RoboDK station: pega_analisa_e_posiciona.rdk

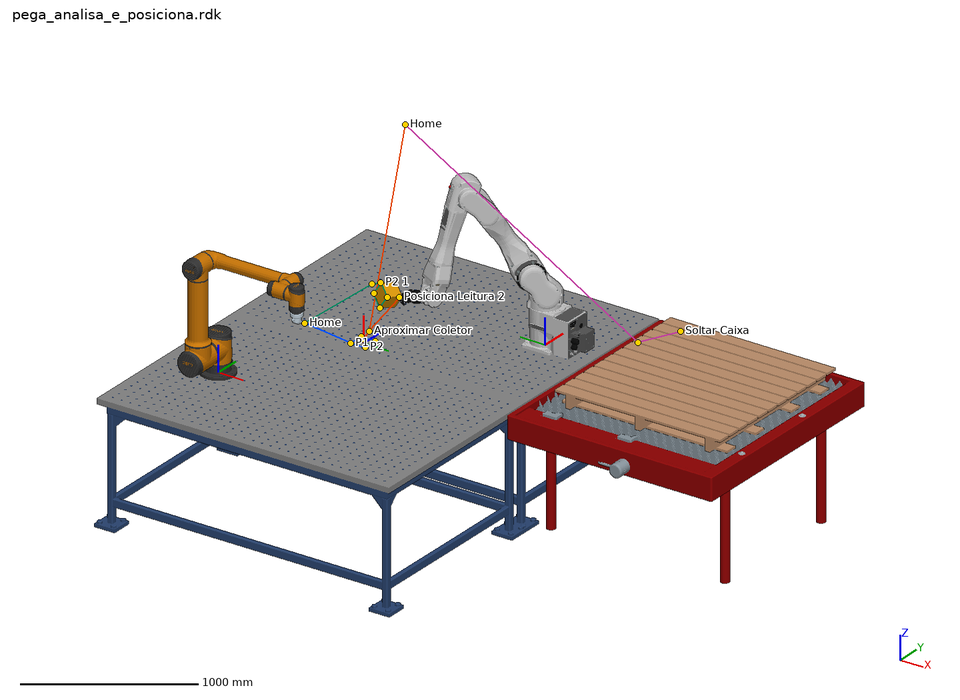
[picture v0: the station drawn from its stored meshes, robots at their saved joint values, targets as dots, program paths as lines]
Station pega_analisa_e_posiciona (saved by RoboDK 6.0.4). Poses are relative to the parent item; angles as X-Y-Z fixed-axis rotations.
  - frame Frame 3 at (0, 2000, 0) mm
    - object Table 2000x1200x800mm at (0, 1320, 0) mm, size 2020 x 1340 x 800 mm, geometry from Table-2000x1200x800mm.sld
    - frame Epson C12XL-A1401 Base at (1300, 1340, 0) mm, rotated rx 0 ry 0 rz 90 deg
      - robot Epson C12XL-A1401: 6 axes, payload 12 kg, reach 1400 mm, repeatability 0.05 mm, weight 63 kg
          modified DH rows (alpha deg, a mm, theta deg, d mm): 0, 0, 0, 472; -90, 100, -90, 0; 0, 650, 0, 0; -90, 30, 0, 650; 90, 0, 0, 0; -90, 0, 0, 80
          base shift (0, 0, 0) mm, rotated rx 0 ry 0 rz 90 deg
          joint limits [-240, -135, -61, -200, -135, -360] to [240, 55, 202, 200, 135, 360]; home [0, 0, 0, 0, 0, 0]; saved at [50.484, -33.978, -40.743, -165.581, -86.297, 207.645]
        - tool RobotiQ 2F-85 Gripper (Fully Closed), TCP at (0, 0, 130) mm, size 121.5 x 75 x 160.2 mm
          - object Cube 100mm at (-37.7, -36.52, 125.42) mm, rotated rx 179.99 ry 0 rz 90 deg, size 100 x 100 x 100 mm, geometry from Cube-100mm.sld
      - target Home (Cartesian target) at (0, 957.19, 1106.49) mm, rotated rx 0 ry -90 rz -90 deg; joints [0, 0, 0, 0, 0, 0] of Epson C12XL-A1401
      - target Aproximar Coletor (Cartesian target) at (-715.16, 704.59, 174.52) mm, rotated rx -180 ry 0 rz 90 deg; joints [43.634, -51.802, 0.005, -180, 38.203, 136.366] of Epson C12XL-A1401
      - target Pegar Caixa (Cartesian target) at (-728.64, 732.29, 119.95) mm, rotated rx -180 ry 0 rz 90 deg; joints [44.857, -55.147, 0.396, -180, 35.249, 135.143] of Epson C12XL-A1401
      - target Posiciona Leitura 2 (Cartesian target) at (-698.85, 508.77, 432.29) mm, rotated rx 69.42 ry -56.81 rz -97.4 deg; joints [50.484, -33.978, -40.743, -165.581, -86.297, 207.645] of Epson C12XL-A1401
      - target Soltar Caixa (Cartesian target) at (172.96, -804.57, 239.71) mm, rotated rx -179.23 ry -0.38 rz -0.85 deg; joints [191.994, -35.632, -24.812, -1.078, -30.231, 78.088] of Epson C12XL-A1401
      - target Aproximar ao local de soltar (Cartesian target) at (-234.04, -797.15, 330.78) mm, rotated rx -179.23 ry -0.38 rz -0.85 deg; joints [163.598, -29.125, -23.601, -0.257, -38.123, 105.753] of Epson C12XL-A1401
    - frame AUBO-i12 Base at (0, 0, 0) mm
      - robot AUBO-i12: 6 axes
          modified DH rows (alpha deg, a mm, theta deg, d mm): 0, 0, 0, 163; 90, 0, 90, 0; 0, 580, 0, 0; 0, 552.5, -90, 191; -90, 0, 0, 117.5; 90, 0, 0, 103.5
          joint limits [-360, -360, -360, -360, -360, -360] to [360, 360, 360, 360, 360, 360]; home [0, 0, 90, 0, 90, 0]; saved at [0, 0, 90, 0, 90, 0]
        - tool Generic Pencil Tool, TCP at (82.2, 0, 101.78) mm, rotated rx 0 ry 60 rz 0 deg, size 125 x 74.9 x 107.3 mm
      - target Home (Cartesian target) at (670, -108.8, 537.72) mm, rotated rx 180 ry -60 rz 90 deg; joints [0, 0, 90, 0, 90, 0] of AUBO-i12
      - target P1 (Cartesian target) at (505.41, 574.84, 94.52) mm, rotated rx 180 ry 0 rz 90 deg; joints [67.254, -32.825, 87.92, -27.207, 70.437, 78.161] of AUBO-i12
      - target P2 (Cartesian target) at (605.41, 574.84, 94.53) mm, rotated rx 180 ry 0 rz 90 deg; joints [61.404, -38.175, 79.011, -29.487, 65.512, 74.753] of AUBO-i12
      - target P3 (Cartesian target) at (605.41, 674.84, 94.52) mm, rotated rx -180 ry 0 rz 90 deg; joints [64.15, -45.805, 65.426, -36.088, 67.815, 76.383] of AUBO-i12
      - target P4 (Cartesian target) at (505.41, 674.84, 94.52) mm, rotated rx 180 ry 0 rz 90 deg; joints [69.61, -40.383, 74.951, -33.036, 72.438, 79.472] of AUBO-i12
      - target P2 3 (Cartesian target) at (745.77, 515.7, 406.16) mm, rotated rx 131.87 ry -73.25 rz 114.52 deg; joints [45.497, -12.081, 99.539, 43.555, 86.097, 65.076] of AUBO-i12
      - target P2 2 (Cartesian target) at (800.05, 508.65, 489.85) mm, rotated rx 131.87 ry -73.25 rz 114.52 deg; joints [42.303, -13.952, 88.161, 34.22, 87.295, 62.11] of AUBO-i12
      - target P2 1 (Cartesian target) at (726.89, 553.6, 541.09) mm, rotated rx 131.87 ry -73.25 rz 114.52 deg; joints [48.541, -9.127, 88.541, 29.382, 84.965, 67.911] of AUBO-i12
      - target P2 4 (Cartesian target) at (672.61, 560.66, 457.4) mm, rotated rx 131.87 ry -73.25 rz 114.52 deg; joints [52.186, -6.843, 99.987, 38.206, 83.627, 71.317] of AUBO-i12
      - target Aproximar 2 (Cartesian target) at (722.97, 468.67, 566.03) mm, rotated rx 131.87 ry -73.25 rz 114.52 deg; joints [44.124, -4.015, 91.726, 27.758, 86.611, 63.8] of AUBO-i12
    - object Table 1500x1400x785mm (Laser Cutting) at (2340, 1230, 0) mm, size 1400 x 1590 x 795.6 mm, geometry from Table-1500x1400x785mm-Laser-Cutting.sld
    - object Table 2000x1200x800mm at (0, 0, 0) mm, size 2020 x 1340 x 800 mm, geometry from Table-2000x1200x800mm.sld
    - object Pallet 1130x1130mm at (1800, 720, 110) mm, size 1130 x 1130.1 x 110 mm, geometry from Pallet-1130x1130mm.sld
  - frame Caixa at (565.41, 2614.84, 94.53) mm, rotated rx 0 ry -90 rz -90 deg
  - program Replace (1 instructions, listed below)
  - program Leitura 1 (9 instructions, listed below)
  - program Pegar Caixa (7 instructions, listed below)
  - program Leitura 2 (10 instructions, listed below)
  - program Soltar Caixa (7 instructions, listed below)
  - program MainProgram (5 instructions, listed below)
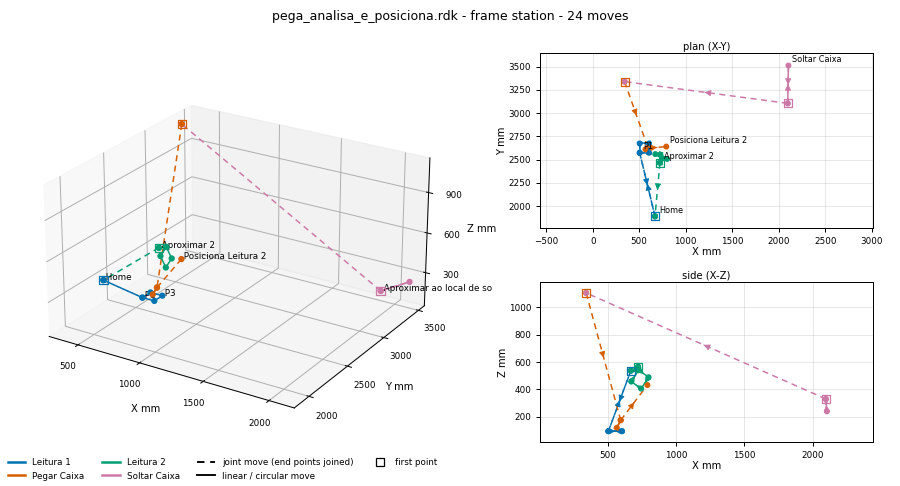
[picture p0: tool path of pega_analisa_e_posiciona.rdk in frame station, 24 of 24 moves have a stored position in this frame; points joined in program order, loops and branches not executed]

--- program Replace (robot Epson C12XL-A1401) ---
  Move objects

--- program Leitura 1 (robot AUBO-i12) ---
  Set Ref.: AUBO-i12 Base
  Set Tool: Generic Pencil Tool
  MoveJ (Home)
  MoveJ (P1)
  MoveL (P2)
  MoveL (P3)
  MoveL (P4)
  MoveL (P1)
  MoveJ (Home)

--- program Pegar Caixa (robot Epson C12XL-A1401) ---
  Set Ref.: Epson C12XL-A1401 Base
  MoveJ (Home)
  MoveJ (Aproximar Coletor)
  MoveL (Pegar Caixa)
  Attach to RobotiQ 2F-85 Gripper (Fully Closed)
  MoveL (Aproximar Coletor)
  MoveJ (Posiciona Leitura 2)

--- program Leitura 2 (robot AUBO-i12) ---
  Set Ref.: AUBO-i12 Base
  Set Tool: Generic Pencil Tool
  MoveJ (Aproximar 2)
  MoveJ (P2 1)
  MoveL (P2 2)
  MoveL (P2 3)
  MoveL (P2 4)
  MoveL (P2 1)
  MoveL (Aproximar 2)
  MoveJ (Home)

--- program Soltar Caixa (robot Epson C12XL-A1401) ---
  Set Ref.: Epson C12XL-A1401 Base
  Set Tool: RobotiQ 2F-85 Gripper (Fully Closed)
  MoveJ (Aproximar ao local de soltar)
  MoveJ (Soltar Caixa)
  Detach from RobotiQ 2F-85 Gripper (Fully Closed)
  MoveL (Aproximar ao local de soltar)
  MoveJ (Home)

--- program MainProgram (robot Epson C12XL-A1401) ---
  Call Replace
  Call Leitura 1
  Call Pegar Caixa
  Call Leitura 2
  Call Soltar Caixa
